FUNCTION_BLOCK Lightspeed EXTENDS PlcModule
VAR_INPUT
	
	{attribute 'OPC.UA.DA' := '0'}
	LightspeedConfig : LightspeedConfig;
	
	{attribute 'OPC.UA.DA' := '0'}
	LsCalibrateConfig : LsCalibrateConfig;
	
	(* Chamber *)
	Chamber : LightspeedChamber(Config := LightspeedConfig.ChamberConfigs.LightspeedChamberConfig);
		
	(* AttenuationFilterConfigs *) 
	FW212CAttenuationFilter : FW212CAttenuationFilter(Config := LightspeedConfig.AttenuationFilterConfigs.FW212CAttenuationFilterConfig);
	ELL14KAttenuationFilter : ELL14KAttenuationFilter(Config := LightspeedConfig.AttenuationFilterConfigs.ELL14KAttenuationFilterConfig);
	ELL9AttenuationFilter : ELL9AttenuationFilter(Config := LightspeedConfig.AttenuationFilterConfigs.ELL9AttenuationFilterConfig);
	
	(* Slider Attenuation *)
	ELL6SliderAttenuationFilter : ELL6AttenuationFilter(Config := LightspeedConfig.SliderAttenuationFilterConfigs.ELL6SliderFilterConfig);													
	
	(* Rotating switch *) 
	ELL18RotatingSwitch : ELL18AttenuationFilter(Config := LightspeedConfig.RotatingSwitchConfigs.ELL18RotatingSwitchConfig);
	
	(* PolarisationFilterConfigs *) 
	FW212CPolarisationFilter : FW212CPolarisationFilter(Config := LightspeedConfig.PolarisationFilterConfigs.FW212CPolarisationFilterConfig);
	ELL14KPolarisationFilter : ELL14KPolarisationFilter(Config := LightspeedConfig.PolarisationFilterConfigs.ELL14KPolarisationFilterConfig, 
														HsPolarisationConfig := LsCalibrateConfig.HSPowermeter.PolarisationConfig,
														HtPolarisationConfig := LsCalibrateConfig.HTPowermeter.PolarisationConfig);
		
	
	(* LaserConfigs *) 
	SMD12Laser : SMD12Laser(Config := LightspeedConfig.LaserConfigs.SMD12LaserConfig);
	Sapphire488Laser : Sapphire488Laser(Config := LightspeedConfig.LaserConfigs.Sapphire488LaserConfig);
	
	(* FiberSwitchConfigs *) 
	EOLFiberSwitch : EOLFiberSwitch(Config := LightspeedConfig.FiberSwitchConfigs.EOLFiberSwitchConfig);
	
	(* OpticalPowermeterConfigs *) 
	PM101OpticalPowermeterHs : PM101OpticalPowermeterHs(Config := LightspeedConfig.OpticalPowermeterConfigs.PM101OpticalPowermeterConfigHs, 
														PolarisationConfig := LsCalibrateConfig.HSPowermeter.PolarisationConfig,
														RFactorSettings := LsCalibrateConfig.HSPowermeter.RFactorSettings,
														ResponsivityConfig := LsCalibrateConfig.HSPowermeter.ResponsivityConfig);
	PM101OpticalPowermeterHt : PM101OpticalPowermeterHt(Config := LightspeedConfig.OpticalPowermeterConfigs.PM101OpticalPowermeterConfigHt, 
														PolarisationConfig := LsCalibrateConfig.HTPowermeter.PolarisationConfig, 
														RFactorSettings := LsCalibrateConfig.HTPowermeter.RFactorSettings,
														ResponsivityConfig := LsCalibrateConfig.HTPowermeter.ResponsivityConfig);
	
	(* DistanceSensorConfigs *) 
	MicroEpsilonDistanceSensor : MicroEpsilonDistanceSensor(Config := LightspeedConfig.DistanceSensorConfigs.MicroEpsilonDistanceSensorConfig);
	
	(* MppcConfigs *) 
	C13336MppcWide   : C13336MppcWide(Config := LightspeedConfig.MppcConfigs.C13336MppcConfigWide);
	C13336MppcNarrow : C13366MppcNarrow(Config := LightspeedConfig.MppcConfigs.C13336MppcConfigNarrow);
	
	(* ShutterConfigs *)
	Ed12dssShutter : Ed12dssShutter(Config := LightspeedConfig.ShutterConfigs.Ed12dssShutterConfig);
	Sh10pilShutter : Sh10pilShutter(Config := LightspeedConfig.ShutterConfigs.Sh10pilShutterConfig);
	
	(* FastAttenuationConfigs *)
	Std900FastAttenuation : Std900FastAttenuation(Config := LightspeedConfig.FastAttenuationConfigs.Std900FastAttenuationConfig);	
	
END_VAR
VAR_OUTPUT
END_VAR
VAR
	{attribute 'OPC.UA.DA' := '0'}
	_startCycling : BOOL;
	{attribute 'OPC.UA.DA' := '0'}
	_count : UINT;
	{attribute 'OPC.UA.DA' := '0'}
	_ActivateCyclingMotorOpen : BOOL ; (* 0 = close door ; 1 = open door  *) 
	{attribute 'OPC.UA.DA' := '0'}
	_CyclingCounterReachSetpoint : BOOL ;
	{attribute 'OPC.UA.DA' := '0'}
	OpenCloseCyclingCount : WORD := 10; (* default value *) 
	{attribute 'OPC.UA.DA' := '0'}
	OpenCloseCurrentCounterValue : WORD:= 0; (* init value *)  ;
	{attribute 'OPC.UA.DA' := '0'}
	WaitingTimer : TON;
	{attribute 'OPC.UA.DA' := '0'}
	DoorSlitOpenCloseCounter: CTU;
	{attribute 'OPC.UA.DA' := '0'}
	OpenCloseCyclingCounterReset : BOOL := FALSE; 
	{attribute 'OPC.UA.DA' := '0'}
	_stopCycling: BOOL:= FALSE;	
	
	{attribute 'OPC.UA.DA' := '0'}
	_mppcActivate : BOOL := TRUE; //TODO à remettre 
	
END_VAR


SUPER^();

IF LightspeedConfig.ChamberConfigs.LightspeedChamberConfig.IsEnabled THEN
	Chamber(MppcActivate => _mppcActivate);	
	
	Door_Slit_Ctrl();
	OpenCloseCycling(_startCycling, _count);
	StopCycling(_stopCycling);	
END_IF

(* Attenuation *)
IF LightspeedConfig.AttenuationFilterConfigs.FW212CAttenuationFilterConfig.IsEnabled THEN		
	FW212CAttenuationFilter();
	IF FW212CAttenuationFilter.InitConfigSerialCom THEN
		;
	END_IF
ELSIF LightspeedConfig.AttenuationFilterConfigs.ELL14KAttenuationFilterConfig.IsEnabled THEN		
	ELL14KAttenuationFilter();
	IF ELL14KAttenuationFilter.InitConfigSerialCom THEN
		;
	END_IF
ELSIF LightspeedConfig.AttenuationFilterConfigs.ELL9AttenuationFilterConfig.IsEnabled THEN		
	ELL9AttenuationFilter();
	IF ELL9AttenuationFilter.InitConfigSerialCom THEN
		;
	END_IF		
END_IF

(* Slider Attenuation *)
IF LightspeedConfig.Version = '2' THEN
	IF LightspeedConfig.SliderAttenuationFilterConfigs.ELL6SliderFilterConfig.IsEnabled THEN		
		ELL6SliderAttenuationFilter();
		IF ELL6SliderAttenuationFilter.InitConfigSerialCom THEN
			;
		END_IF
	END_IF
END_IF

(* Rotating switch *)
IF LightspeedConfig.Version = '2' THEN
	IF LightspeedConfig.RotatingSwitchConfigs.ELL18RotatingSwitchConfig.IsEnabled THEN		
		ELL18RotatingSwitch();
		IF ELL18RotatingSwitch.InitConfigSerialCom THEN
			;
		END_IF
	END_IF
END_IF

IF LightspeedConfig.PolarisationFilterConfigs.FW212CPolarisationFilterConfig.IsEnabled THEN
	FW212CPolarisationFilter();	
	IF FW212CPolarisationFilter.InitConfigSerialCom THEN
		;
	END_IF
ELSIF LightspeedConfig.PolarisationFilterConfigs.ELL14KPolarisationFilterConfig.IsEnabled THEN		
	ELL14KPolarisationFilter();
	IF ELL14KPolarisationFilter.InitConfigSerialCom THEN
		;
	END_IF			
END_IF

IF LightspeedConfig.LaserConfigs.SMD12LaserConfig.IsEnabled THEN
	SMD12Laser();
	IF SMD12Laser.InitConfigSerialCom THEN
		;
	END_IF
ELSIF LightspeedConfig.LaserConfigs.Sapphire488LaserConfig.IsEnabled THEN
	Sapphire488Laser();
	IF Sapphire488Laser.InitConfigSerialCom THEN
		;
	END_IF
ELSIF LightspeedConfig.LaserConfigs.Sapphire488LaserConfig.IsEnabled THEN
	Sapphire488Laser();
	IF Sapphire488Laser.InitConfigSerialCom THEN
		;
	END_IF	
END_IF

IF LightspeedConfig.FiberSwitchConfigs.EOLFiberSwitchConfig.IsEnabled THEN
	EOLFiberSwitch();
	IF EOLFiberSwitch.InitConfigSerialCom THEN
		;
	END_IF
END_IF

IF LightspeedConfig.OpticalPowermeterConfigs.PM101OpticalPowermeterConfigHs.IsEnabled OR 
   LightspeedConfig.OpticalPowermeterConfigs.PM101OpticalPowermeterConfigHs.IsSimulated THEN
	PM101OpticalPowermeterHs(PolarResult := ELL14KPolarisationFilter.PolarResult);
	IF PM101OpticalPowermeterHs.InitConfigSerialCom THEN
		;
	END_IF	
END_IF

IF LightspeedConfig.OpticalPowermeterConfigs.PM101OpticalPowermeterConfigHt.IsEnabled THEN
	PM101OpticalPowermeterHt(PolarResult := ELL14KPolarisationFilter.PolarResult);
	IF PM101OpticalPowermeterHt.InitConfigSerialCom THEN
		;
	END_IF	
END_IF

IF LightspeedConfig.DistanceSensorConfigs.MicroEpsilonDistanceSensorConfig.IsEnabled THEN
	MicroEpsilonDistanceSensor();	
END_IF

IF LightspeedConfig.MppcConfigs.C13336MppcConfigWide.IsEnabled THEN
	C13336MppcWide(MppcActivate := _mppcActivate);
	IF C13336MppcWide.InitConfigSerialCom THEN
		;
	END_IF
END_IF

IF LightspeedConfig.MppcConfigs.C13336MppcConfigNarrow.IsEnabled THEN
	C13336MppcNarrow(MppcActivate := _mppcActivate);
	IF C13336MppcNarrow.InitConfigSerialCom THEN
		;
	END_IF
END_IF

IF LightspeedConfig.ShutterConfigs.Ed12dssShutterConfig.IsEnabled THEN
	Ed12dssShutter();	
ELSIF LightspeedConfig.ShutterConfigs.SH10PILShutterConfig.IsEnabled THEN
	Sh10pilShutter();
END_IF

IF LightspeedConfig.FastAttenuationConfigs.Std900FastAttenuationConfig.IsEnabled THEN
	Std900FastAttenuation();	
END_IF

METHOD Door_Slit_Ctrl : BOOL
VAR_INPUT	
END_VAR
VAR
	timeout : TIME := T#1400MS; (* 2 * open time (700ms)  *) 
	MotorTurnOffAfterTimeout: TON;
END_VAR
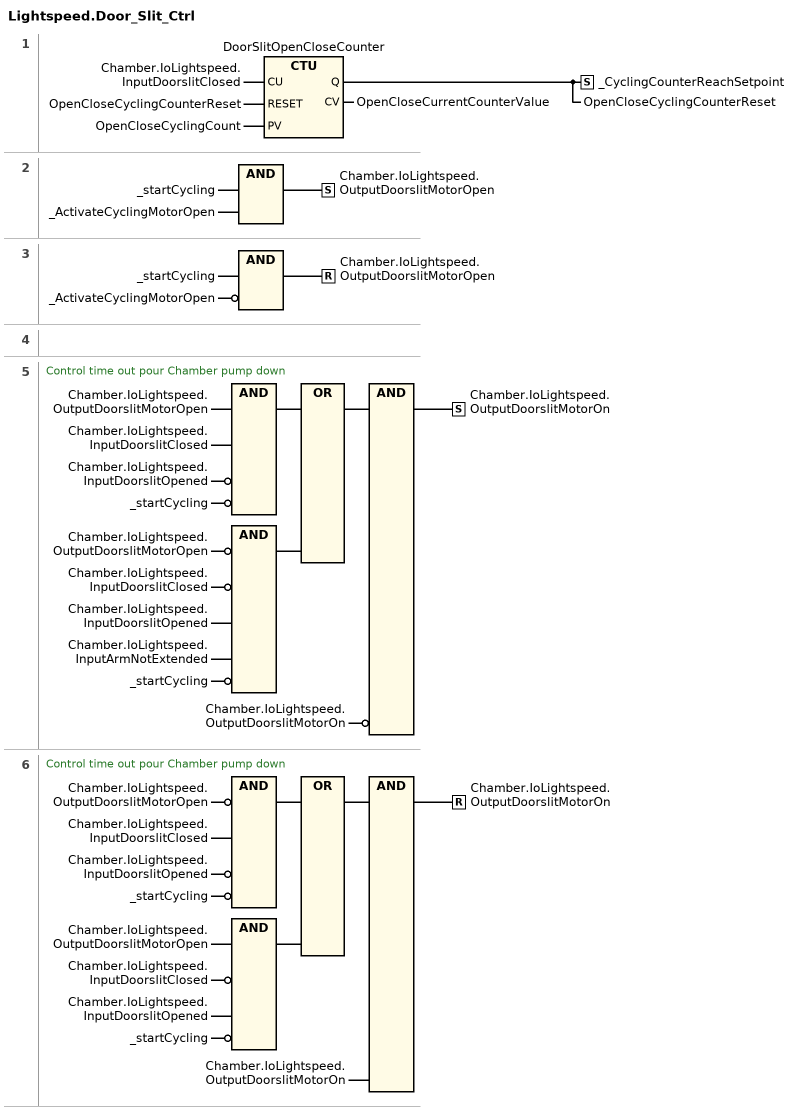
// NETWORK 1
DoorSlitOpenCloseCounter(
    CU := Chamber.IoLightspeed.InputDoorslitClosed,
    RESET := OpenCloseCyclingCounterReset,
    PV := OpenCloseCyclingCount,
    CV => OpenCloseCurrentCounterValue); // CTU
_CyclingCounterReachSetpoint S= DoorSlitOpenCloseCounter.Q;
OpenCloseCyclingCounterReset := DoorSlitOpenCloseCounter.Q;

// NETWORK 2
Chamber.IoLightspeed.OutputDoorslitMotorOpen S= _startCycling AND _ActivateCyclingMotorOpen;

// NETWORK 3
Chamber.IoLightspeed.OutputDoorslitMotorOpen R= _startCycling AND NOT _ActivateCyclingMotorOpen;

// NETWORK 4

// NETWORK 5
// Control time out pour Chamber pump down
Chamber.IoLightspeed.OutputDoorslitMotorOn S= (Chamber.IoLightspeed.OutputDoorslitMotorOpen AND Chamber.IoLightspeed.InputDoorslitClosed AND NOT Chamber.IoLightspeed.InputDoorslitOpened AND NOT _startCycling OR NOT Chamber.IoLightspeed.OutputDoorslitMotorOpen AND NOT Chamber.IoLightspeed.InputDoorslitClosed AND Chamber.IoLightspeed.InputDoorslitOpened AND Chamber.IoLightspeed.InputArmNotExtended AND NOT _startCycling) AND NOT Chamber.IoLightspeed.OutputDoorslitMotorOn;

// NETWORK 6
// Control time out pour Chamber pump down
Chamber.IoLightspeed.OutputDoorslitMotorOn R= (NOT Chamber.IoLightspeed.OutputDoorslitMotorOpen AND Chamber.IoLightspeed.InputDoorslitClosed AND NOT Chamber.IoLightspeed.InputDoorslitOpened AND NOT _startCycling OR Chamber.IoLightspeed.OutputDoorslitMotorOpen AND NOT Chamber.IoLightspeed.InputDoorslitClosed AND Chamber.IoLightspeed.InputDoorslitOpened AND NOT _startCycling) AND Chamber.IoLightspeed.OutputDoorslitMotorOn;

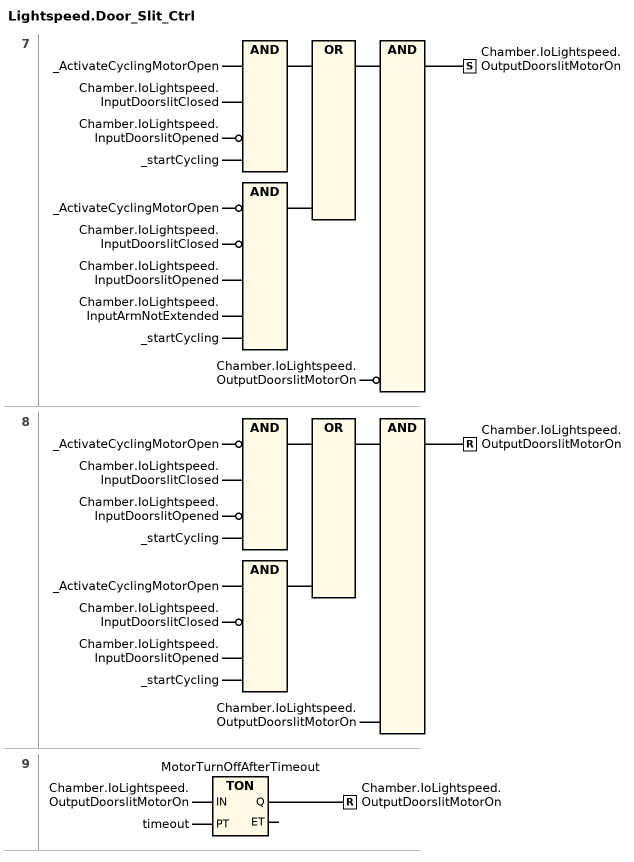
// NETWORK 7
Chamber.IoLightspeed.OutputDoorslitMotorOn S= (_ActivateCyclingMotorOpen AND Chamber.IoLightspeed.InputDoorslitClosed AND NOT Chamber.IoLightspeed.InputDoorslitOpened AND _startCycling OR NOT _ActivateCyclingMotorOpen AND NOT Chamber.IoLightspeed.InputDoorslitClosed AND Chamber.IoLightspeed.InputDoorslitOpened AND Chamber.IoLightspeed.InputArmNotExtended AND _startCycling) AND NOT Chamber.IoLightspeed.OutputDoorslitMotorOn;

// NETWORK 8
Chamber.IoLightspeed.OutputDoorslitMotorOn R= (NOT _ActivateCyclingMotorOpen AND Chamber.IoLightspeed.InputDoorslitClosed AND NOT Chamber.IoLightspeed.InputDoorslitOpened AND _startCycling OR _ActivateCyclingMotorOpen AND NOT Chamber.IoLightspeed.InputDoorslitClosed AND Chamber.IoLightspeed.InputDoorslitOpened AND _startCycling) AND Chamber.IoLightspeed.OutputDoorslitMotorOn;

// NETWORK 9
MotorTurnOffAfterTimeout(IN := Chamber.IoLightspeed.OutputDoorslitMotorOn, PT := timeout); // TON
Chamber.IoLightspeed.OutputDoorslitMotorOn R= MotorTurnOffAfterTimeout.Q;
END_METHOD

METHOD FB_init : BOOL
VAR_INPUT
	bInitRetains : BOOL; // if TRUE, the retain variables are initialized (warm start / cold start)
	bInCopyCode : BOOL;  // if TRUE, the instance afterwards gets moved into the copy code (online change)
	Config : LightspeedConfig;
	CalibrateConfig : LsCalibrateConfig;
END_VAR
LightspeedConfig := Config;
LsCalibrateConfig := CalibrateConfig;
LsBkgrdLsSerialCom(Config := LightspeedConfig);

IF Config.IsEnabled THEN
	_logger.Information('Lightspeed devices initialization starting...');
END_IF	

(* Chamber *)
IF Config.ChamberConfigs.LightspeedChamberConfig.IsEnabled THEN
	Chamber.FB_init(FALSE, FALSE, Config := Config.ChamberConfigs.LightspeedChamberConfig);	
END_IF

(* AttenuationFilterConfigs *)
IF Config.AttenuationFilterConfigs.FW212CAttenuationFilterConfig.IsEnabled THEN
	FW212CAttenuationFilter.FB_init(FALSE, FALSE, Config := Config.AttenuationFilterConfigs.FW212CAttenuationFilterConfig);	
ELSIF Config.AttenuationFilterConfigs.ELL14KAttenuationFilterConfig.IsEnabled THEN
	ELL14KAttenuationFilter.FB_init(FALSE, FALSE, Config := Config.AttenuationFilterConfigs.ELL14KAttenuationFilterConfig);
END_IF

(* Slider Attenuation *)
IF Config.Version = '2' THEN
	IF Config.SliderAttenuationFilterConfigs.ELL6SliderFilterConfig.IsEnabled THEN
		ELL6SliderAttenuationFilter.FB_init(FALSE, FALSE, Config := Config.SliderAttenuationFilterConfigs.ELL6SliderFilterConfig);
	END_IF
END_IF

(* Rotating switch *)
IF Config.Version = '2' THEN
	IF Config.RotatingSwitchConfigs.ELL18RotatingSwitchConfig.IsEnabled THEN
		ELL18RotatingSwitch.FB_init(FALSE, FALSE, Config := Config.RotatingSwitchConfigs.ELL18RotatingSwitchConfig);
	END_IF
END_IF

(* PolarisationFilterConfigs *)
IF Config.PolarisationFilterConfigs.FW212CPolarisationFilterConfig.IsEnabled THEN
	FW212CPolarisationFilter.FB_init(FALSE, FALSE, Config := Config.PolarisationFilterConfigs.FW212CPolarisationFilterConfig);	
ELSIF Config.PolarisationFilterConfigs.ELL14KPolarisationFilterConfig.IsEnabled THEN
	ELL14KPolarisationFilter.FB_init(FALSE, FALSE, Config := Config.PolarisationFilterConfigs.ELL14KPolarisationFilterConfig, 
												   HsPolarisationConfig := CalibrateConfig.HSPowermeter.PolarisationConfig,
												   HtPolarisationConfig := CalibrateConfig.HTPowermeter.PolarisationConfig);
END_IF

(* LaserConfigs *) 
IF Config.LaserConfigs.SMD12LaserConfig.IsEnabled THEN
	SMD12Laser.FB_init(FALSE, FALSE, Config := Config.LaserConfigs.SMD12LaserConfig);	
ELSIF Config.LaserConfigs.Sapphire488LaserConfig.IsEnabled THEN
	Sapphire488Laser.FB_init(FALSE, FALSE, Config := Config.LaserConfigs.Sapphire488LaserConfig);	
END_IF

(* FiberSwitchConfigs *) 
IF Config.FiberSwitchConfigs.EOLFiberSwitchConfig.IsEnabled THEN
	EOLFiberSwitch.FB_init(FALSE, FALSE, Config := Config.FiberSwitchConfigs.EOLFiberSwitchConfig);	
END_IF

(* OpticalPowermeterConfigs *) 
IF Config.OpticalPowermeterConfigs.PM101OpticalPowermeterConfigHs.IsEnabled THEN
	PM101OpticalPowermeterHs.FB_init(FALSE, FALSE, Config := Config.OpticalPowermeterConfigs.PM101OpticalPowermeterConfigHs, 
												   PolarisationConfig := CalibrateConfig.HSPowermeter.PolarisationConfig, 
												   RFactorSettings := CalibrateConfig.HSPowermeter.RFactorSettings,
												   ResponsivityConfig := CalibrateConfig.HSPowermeter.ResponsivityConfig);		
END_IF
IF Config.OpticalPowermeterConfigs.PM101OpticalPowermeterConfigHt.IsEnabled THEN
	PM101OpticalPowermeterHt.FB_init(FALSE, FALSE, Config := Config.OpticalPowermeterConfigs.PM101OpticalPowermeterConfigHt, 
												   PolarisationConfig := CalibrateConfig.HTPowermeter.PolarisationConfig,
												   RFactorSettings := CalibrateConfig.HTPowermeter.RFactorSettings,
												   ResponsivityConfig := CalibrateConfig.HTPowermeter.ResponsivityConfig);
END_IF

(* DistanceSensorConfigs *) 
IF Config.DistanceSensorConfigs.MicroEpsilonDistanceSensorConfig.IsEnabled THEN
	MicroEpsilonDistanceSensor.FB_init(FALSE, FALSE, Config := Config.DistanceSensorConfigs.MicroEpsilonDistanceSensorConfig);	
END_IF

(* MppcConfigs *) 
IF Config.MppcConfigs.C13336MppcConfigWide.IsEnabled THEN
	C13336MppcWide.FB_init(FALSE, FALSE, Config := Config.MppcConfigs.C13336MppcConfigWide);	
END_IF
IF Config.MppcConfigs.C13336MppcConfigNarrow.IsEnabled THEN
	C13336MppcNarrow.FB_init(FALSE, FALSE, Config := Config.MppcConfigs.C13336MppcConfigNarrow);	
END_IF

(* ShutterConfigs *) 
IF Config.ShutterConfigs.Ed12dssShutterConfig.IsEnabled THEN
	Ed12dssShutter.FB_init(FALSE, FALSE, Config := Config.ShutterConfigs.Ed12dssShutterConfig);	
ELSIF Config.ShutterConfigs.SH10PILShutterConfig.IsEnabled THEN
	Sh10pilShutter.FB_init(FALSE, FALSE, Config := Config.ShutterConfigs.SH10PILShutterConfig);	
END_IF

IF Config.IsEnabled THEN
	_logger.Information('Lightspeed devices initialization ended...');
END_IF
END_METHOD

METHOD OpenCloseCycling : BOOL
VAR_INPUT
	Execute : BOOL;
	Count : UINT;
END_VAR
VAR 
END_VAR
IF Execute THEN
	(* timer pour l'enchainement des open/close *)
	(* WaitingTimer.in := TRUE;
	WaitingTimer.PT := T#4S;*)
	WaitingTimer (IN :=TRUE , PT := T#5S,Q=>, ET=> );
	
	(* WaitingTimer.Q is TRUE, PT seconds after IN had a rising edge *)
	IF WaitingTimer.Q THEN
		(* RAZ du timer *)
		WaitingTimer (IN := FALSE);
		(* coupe le motor ON par securité*)
		Chamber.IoLightspeed.OutputDoorslitMotorOn := FALSE;
		(* MAJ du compteur*)
		OpenCloseCyclingCount := Count;
		(* porte ouverte => on demande la fermeture*)
		IF (_CyclingCounterReachSetpoint) THEN
			(* arret du cycling et re init des variables*)
			Chamber.IoLightspeed.OutputDoorslitMotorOn := FALSE;
			_startCycling := FALSE;
			_CyclingCounterReachSetpoint := FALSE;
			_ActivateCyclingMotorOpen := FALSE;
			OpenCloseCycling := FALSE;
			OpenCloseCurrentCounterValue := 0;
			(* to do lever un timeout vers acquisition si not(_CyclingCounterReachSetpoint) => pb d'open/close  *)
		ELSIF Chamber.IoLightspeed.InputDoorslitOpened THEN
			_ActivateCyclingMotorOpen := FALSE;	
		(* porte fermée => on demande l'ouverture *)			
		ELSIF (Chamber.IoLightspeed.InputDoorslitClosed) THEN
			_ActivateCyclingMotorOpen := TRUE;	
		END_IF
	END_IF
END_IF
END_METHOD

METHOD StopCycling : BOOL
VAR_INPUT
	Execute : BOOL;
END_VAR
VAR 
END_VAR
IF Execute THEN
	(* stop du cycling*)
	(* on attend le porte fermée pour arreter le cycling *)
	IF ( NOT (Chamber.IoLightspeed.InputDoorslitOpened) AND Chamber.IoLightspeed.InputDoorslitClosed)  THEN
		(* arret du cycling et re init des variables*)
		(* arret du cycling *)
		_startCycling := FALSE;
		(* coupe le moteur par securité *)
		Chamber.IoLightspeed.OutputDoorslitMotorOn := FALSE;
		(* fin du stop cycling*)
		_stopCycling:= FALSE;
		(* re init du compteur de cycle *)
		_CyclingCounterReachSetpoint := FALSE;
		OpenCloseCurrentCounterValue := 0;
		OpenCloseCyclingCount := 0;
	END_IF
END_IF
END_METHOD

END_FUNCTION_BLOCK

(* stored: Version 1.1.0.1, ProductVersion 3.1.4024.12
   POU Lightspeed: Id {b1820b5e-8283-43dc-b399-2d75c16eb6f0}, SpecialFunc None
   Folder DoorSlit: Id {7e3189a0-bffc-4d7d-8844-3b5c5fe06446}
   Method Door_Slit_Ctrl: Id {c5558a09-4fa8-46b4-9972-cde4601d6796}
   Method FB_init: Id {09564059-546a-497c-9b54-4b93903ae9de}
   Method OpenCloseCycling: Id {8a380f41-0443-4c66-a6ce-51982bdb92a2}
   Method StopCycling: Id {74208cd1-90d0-4c46-8202-5e5729222b64} *)
